INTERFACE I_State

METHOD PUBLIC Check
END_METHOD

PROPERTY PUBLIC Description : STRING
GET
END_GET
END_PROPERTY

METHOD PUBLIC PressButton
END_METHOD

METHOD PUBLIC PressDischarge
END_METHOD

METHOD PUBLIC Reset
END_METHOD

METHOD PUBLIC Stop
END_METHOD

METHOD PUBLIC TimerDone
END_METHOD

END_INTERFACE

(* stored: Version 1.1.0.1, ProductVersion 3.1.4024.12
   Itf I_State: Id {1bde4dc7-ad40-4977-a870-ea0a6b0033a4}
   Method Check: Id {b245be02-aa95-4793-a4a1-45881f680e36}
   Property Description: Id {0887b0dc-99d1-4e94-a136-582c1cd1dded}
   Get Get: Id {f15343b1-d437-42e5-9325-bf2fc67af358}
   Method PressButton: Id {5f90240b-e852-4d11-809b-01436ec01f56}
   Method PressDischarge: Id {58412862-6253-4565-abcf-db6579e1f705}
   Method Reset: Id {ec94a8f1-7aa1-443c-bd08-21942ad945a8}
   Method Stop: Id {95bfd00f-897b-4976-8d1f-deb515d63881}
   Method TimerDone: Id {bb9a359f-c0ba-4be7-9e53-9cedbe13fd26} *)
